FUNCTION F_IsNumber : BOOL
(*Returns true if the charachter is a number*)
VAR_INPUT
	sChr				: STRING(1);
END_VAR
VAR
END_VAR

F_IsNumber := (F_ToASC(sChr) >= 16#30 AND F_ToASC(sChr) <= 16#39);

END_FUNCTION

(* stored: Version 1.1.0.1
   POU F_IsNumber: Id {be9138be-b37b-4501-8d6e-7e23f70be1bc}, SpecialFunc None *)
